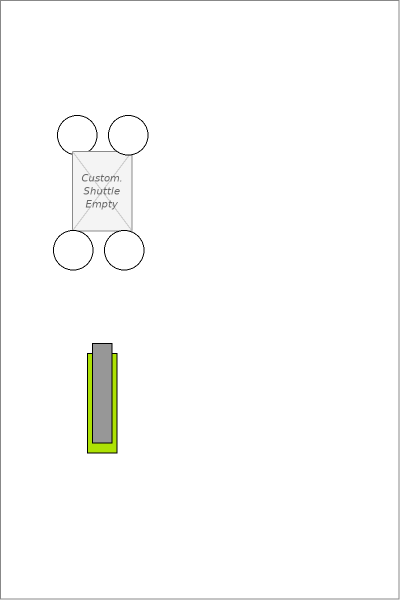
VISUALIZATION VISU_ST175  // 400x600
    Ellipse (57,115 40x40), colour toggle: GVL.st160_aut.fb_ABL_CETA.fb_capMainteningLeft.xIN_AS
    Image (72,151 60x80), angle 90, invisible if: NOT __ISVALIDREF(GVL.st160_aut._Mover), image: Custom.Shuttle Empty
    Ellipse (108,115 40x40), colour toggle: GVL.st160_aut.fb_ABL_CETA.fb_capMainteningRight.xIN_AS
    Rectangle (87,353 30x100)
    Rectangle (92,343 20x100)
        p2738717112: -GVL.st160_aut.fb_ABL_CETA.simu_axis160_01Z.rOUT_PixActual
    Ellipse (53,230 40x40), colour toggle: GVL.st160_aut.fb_ABL_CETA.fb_dichtung_left.xIN_AS
    Ellipse (104,230 40x40), colour toggle: GVL.st160_aut.fb_ABL_CETA.fb_dichtung_right.xIN_AS
END_VISUALIZATION

(* stored: Version 1.1.0.1, ProductVersion 3.1.4024.6
   Visu VISU_ST175: Id {2a3388fe-26aa-499d-80ed-08924182db9d} *)
